// TIA Portal V19 export
VAR_GLOBAL   // PLC tag table "Decoilers_IO"
   DecoilerX_AI_Coil_Diameter AT %IW906 : Int;   // 464A1 - 736BF1
   Decoier1_Coupling_Ls_Rest AT %I125.5 : Bool;   // 710SQ1
   Decoier1_Coupling_Ls_Work AT %I125.6 : Bool;   // 710SQ2
   Decoiler1_Coupling_V_Rest AT %Q100.6 : Bool;   // 710YV1
   Decoiler1_Coupling_V_Work AT %Q100.7 : Bool;   // 710YV2
   Decoiler1_Jaws_V_Close AT %Q101.1 : Bool;   // 711YV1
   Decoiler1_Jaws_V_Open AT %Q101.2 : Bool;   // 711YV2
   Decoiler1_PneuBrake_1_V_Open AT %Q130.0 : Bool;   // 745YV1
   Decoiler1_PneuBrake_1_V_Partial AT %Q130.1 : Bool;   // 745YV1
   Decoiler1_M_Fan_C AT %Q0.7 : Bool;   // 742QF1
   Decoiler1_M_Fan_Fdbk AT %I3.2 : Bool;   // 742KM1
   Decoiler2_Coupling_Ls_Rest AT %I126.0 : Bool;   // 715SQ1
   Decoiler2_Coupling_Ls_Work AT %I126.1 : Bool;   // 715SQ2
   Decoiler2_Coupling_V_Rest AT %Q101.7 : Bool;   // 715YV1
   Decoiler2_Coupling_V_Work AT %Q102.0 : Bool;   // 715YV2
   Decoiler2_Jaws_V_Close AT %Q102.1 : Bool;   // 716YV1
   Decoiler2_Jaws_V_Open AT %Q102.2 : Bool;   // 716YV2
   Decoiler2_PneuBrake_1_V_Open AT %Q130.4 : Bool;   // 755YV1
   Decoiler2_PneuBrake_1_V_Partial AT %Q130.5 : Bool;   // 755YV2
   Decoiler2_M_Fan_C AT %Q1.0 : Bool;   // 752QF1
   Decoiler2_M_Fan_Fdbk AT %I3.3 : Bool;   // 752KM1
   Decoiler1_PneuBrake_2_V_Close AT %Q130.2 : Bool;   // 745YV3
   Decoiler1_PneuBrake_2_V_Partial AT %Q130.3 : Bool;   // 745YV4
   Decoiler2_PneuBrake_2_V_Close AT %Q130.6 : Bool;   // 755YV3
   Decoiler2_PneuBrake_2_V_Partial AT %Q130.7 : Bool;   // 755YV4
   DecoilerX_LIBERO AT %I126.3 : Bool;   // 735 - LIBERO
   DecoilerX_MaterialPresence AT %I126.4 : Bool;   // 735BF1
   DecoilerX_NOT_USED AT %I126.5 : Bool;   // 735BF2
   Decoiler2_PosizioneRazza AT %I142.7 : Bool;
END_VAR
